{attribute addProperty BoxType "KL8610"}
{attribute addProperty Id "KL8601_1KL_B0A8062F00"}
{attribute addProperty CRC "151672865"}
{attribute addProperty SizeInBites "0"}
{attribute addProperty SizeInBytes "0"}
TYPE KL8610_090A5821 :
STRUCT
	{attribute addProperty Name "KL8601_1"}
	KL8601_1 : KL_B0A8062F;
END_STRUCT
END_TYPE

(* stored: Version 1.2.0.0, ProductVersion 3.1.4024.9
   DUT KL8610_090A5821: Id {20834643-6f0f-4887-a826-c6497d00f086} *)
